% RSLogix 500 project Y-AXIS.RSS, saved by version 8.30.00.16 %
PROJECT "UNTITLED"    % processor: Bul.1763 MicroLogix 1100 Series B %

PROGRAM FILES
  LAD 2   8 rungs

DATA FILES
  O0 OUTPUT  5 elements
  I1 INPUT  7 elements
  S2 STATUS  66 elements
  B3 BINARY  2 elements
  T4 TIMER  1 elements
  C5 COUNTER  1 elements
  R6 CONTROL  1 elements
  N7 INTEGER  2 elements
  F8 FLOAT  1 elements

LADDER 2
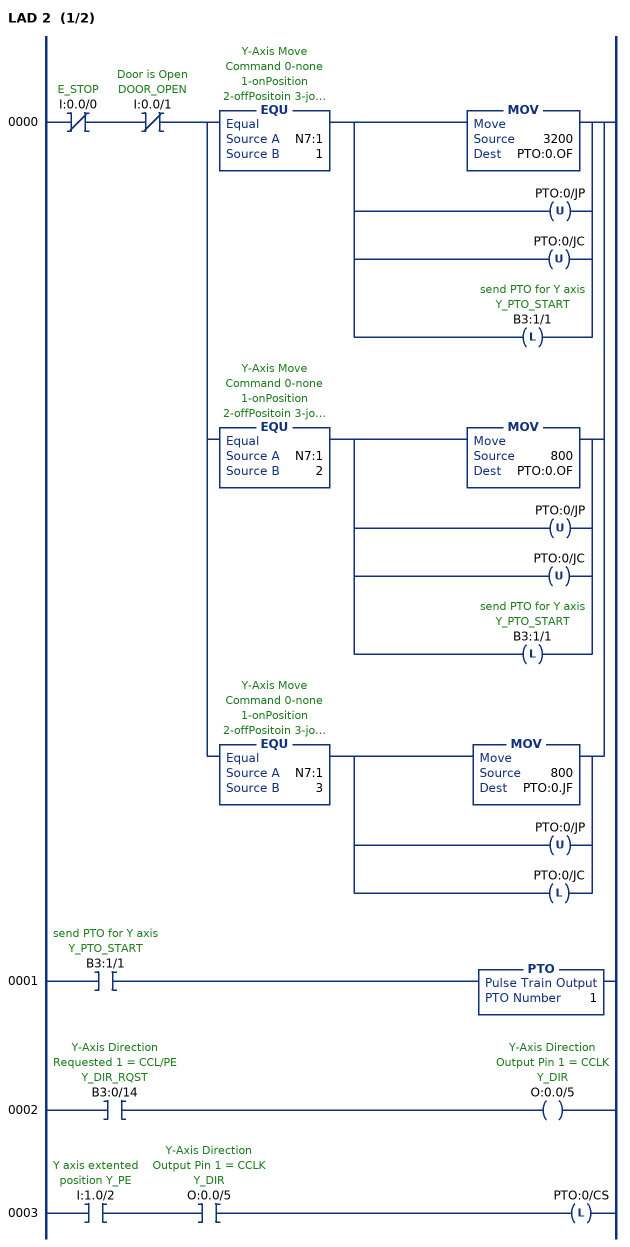
% Rung: 0 %
SOR XIO I:0.0/0 XIO I:0.0/1 BST EQU N7:1 1 BST MOV 3200 PTO:0.OF NXB OTU PTO:0/JP NXB OTU PTO:0/JC NXB OTL B3:1/1 BND NXB EQU N7:1 2 BST MOV 800 PTO:0.OF NXB OTU PTO:0/JP NXB OTU PTO:0/JC NXB OTL B3:1/1 BND NXB EQU N7:1 3 BST MOV 800 PTO:0.JF NXB OTU PTO:0/JP NXB OTL PTO:0/JC BND BND EOR
%   I:0.0/0  E_STOP %
%   I:0.0/1  DOOR_OPEN  "Door is Open" %
%   N7:1  Y_CMD_TYPE  "Y-Axis Move Command 0-none 1-onPosition 2-offPositoin 3-jog" %
%   B3:1/1  Y_PTO_START  "send PTO for Y axis" %
% Rung: 1 %
SOR XIC B3:1/1 PTO 1 EOR
%   B3:1/1  Y_PTO_START  "send PTO for Y axis" %
% Rung: 2 %
SOR XIC B3:0/14 OTE O:0.0/5 EOR
%   B3:0/14  Y_DIR_RQST  "Y-Axis Direction Requested 1 = CCL/PE" %
%   O:0.0/5  Y_DIR  "Y-Axis Direction Output Pin 1 = CCLK" %
% Rung: 3 %
SOR XIC I:1.0/2 XIC O:0.0/5 OTL PTO:0/CS EOR
%   I:1.0/2  Y_PE  "Y axis extented position" %
%   O:0.0/5  Y_DIR  "Y-Axis Direction Output Pin 1 = CCLK" %

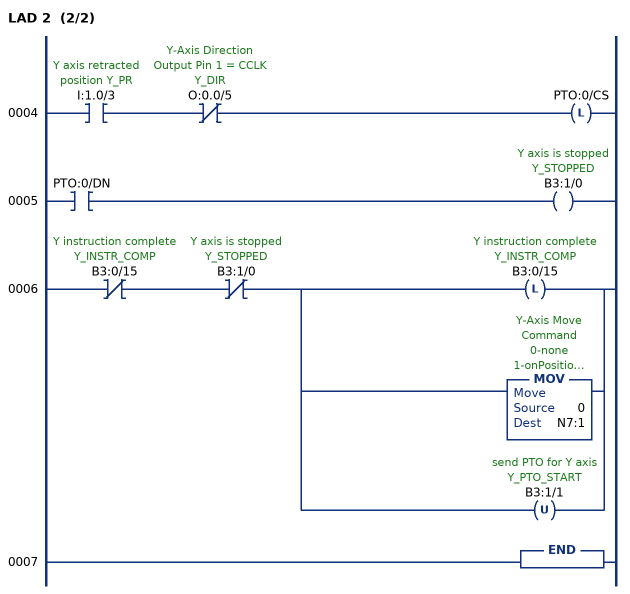
% Rung: 4 %
SOR XIC I:1.0/3 XIO O:0.0/5 OTL PTO:0/CS EOR
%   I:1.0/3  Y_PR  "Y axis retracted position" %
%   O:0.0/5  Y_DIR  "Y-Axis Direction Output Pin 1 = CCLK" %
% Rung: 5 %
SOR XIC PTO:0/DN OTE B3:1/0 EOR
%   B3:1/0  Y_STOPPED  "Y axis is stopped" %
% Rung: 6 %  % edit flag set %
SOR XIO B3:0/15 XIO B3:1/0 BST OTL B3:0/15 NXB MOV 0 N7:1 NXB OTU B3:1/1 BND EOR
%   B3:0/15  Y_INSTR_COMP  "Y instruction complete" %
%   B3:1/0  Y_STOPPED  "Y axis is stopped" %
%   N7:1  Y_CMD_TYPE  "Y-Axis Move Command 0-none 1-onPosition 2-offPositoin 3-jog" %
%   B3:1/1  Y_PTO_START  "send PTO for Y axis" %
% Rung: 7 %
SOR END EOR

OTHER DOCUMENTED ADDRESSES
  PTO:0.1/5  Y_CTRL_STOP  "Controlled Stop Y- Axis"
  PTO:0.3  Y_SPEED  "Y-AXIS MOVE SPEED"
  PTO:0.5  Y_JOG_SPEED  "Y-Axis Jog Speed"
